FUNCTION_BLOCK TwoAlgs
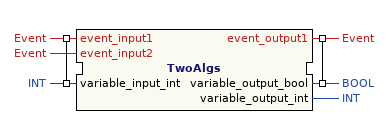
  EVENT_INPUT
    event_input1 WITH variable_input_int;
    event_input2;
  END_EVENT
  EVENT_OUTPUT
    event_output1 WITH variable_output_bool;
  END_EVENT
  VAR_INPUT
    variable_input_int : INT;
  END_VAR
  VAR_OUTPUT
    variable_output_bool : BOOL;
    variable_output_int : INT;
  END_VAR
  VAR
    internal_variable1 : STRING;
  END_VAR
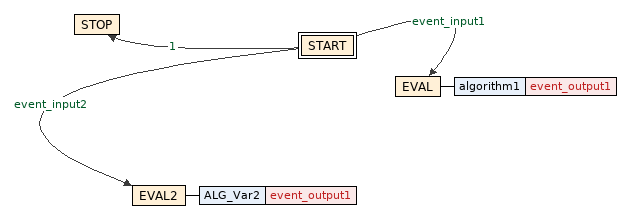
  EC_STATES
    START;
    STOP;
    EVAL : algorithm1 -> event_output1;
    EVAL2 : ALG_Var2 -> event_output1;
  END_STATES
  EC_TRANSITIONS
    START TO STOP := 1;
    START TO EVAL := event_input1;
    START TO EVAL2 := event_input2;
  END_TRANSITIONS
  ALGORITHM algorithm1 IN ST:
  VAR_TEMP
    delta : INT;
  END_VAR
delta := 4;&#38;#10;variable_output_bool := TRUE;&#38;#10;variable_output_int := delta + 7;&#38;#10;
  END_ALGORITHM
  ALGORITHM ALG_Var2 IN ST:
  VAR_TEMP
    tmpVar : BOOL;
    tmpVar2 : STRING;
  END_VAR
tmpVar := TRUE;&#38;#10;tmpVar2 := &#39;novalue&#39;;&#38;#10;variable_output_bool := FALSE;&#38;#10;variable_output_int := 0;&#38;#10;
  END_ALGORITHM
END_FUNCTION_BLOCK
